{attribute 'qualified_only'}
{attribute 'strict'}
TYPE E_MoveAbsoluteMode :
(
	ONLY_MOVE := 0,
	CALC_TIME_START_IMMEDIATELY := 1,
	CALC_TIME_DELAY_START	:= 2
);
END_TYPE

(* stored: Version 1.1.0.1, ProductVersion 3.1.4022.12
   DUT E_MoveAbsoluteMode: Id {8ab523b1-1b56-4f58-9898-0392516727e2} *)
